{attribute 'linkalways'} 
{attribute 'no_explicit_call' := 'This FB is a CLASS and must be accessed using methods or properties'}
{attribute 'enable_dynamic_creation'}
FUNCTION_BLOCK NodeAddedEvent EXTENDS Disposable IMPLEMENTS I_NodeAddedEvent
VAR
	_target : I_Node;
END_VAR

METHOD FB_init : BOOL
VAR_INPUT
	bInitRetains : BOOL; // if TRUE, the retain variables are initialized (warm start / cold start)
	bInCopyCode : BOOL;  // if TRUE, the instance afterwards gets moved into the copy code (online change)
	Target : I_Node;
END_VAR
This^._target := Target;
END_METHOD

PROPERTY PUBLIC Target : I_Node
GET
Target := _target;
END_GET
END_PROPERTY

END_FUNCTION_BLOCK

(* stored: Version 1.1.0.1, ProductVersion 3.1.4024.12
   POU NodeAddedEvent: Id {675de5f9-7ea0-47ea-9f02-f8d732921215}, SpecialFunc None
   Folder Constructor: Id {3f775415-77de-4978-87d9-9c8a995c1d0f}
   Method FB_init: Id {79ddcdd9-31d4-44ed-94b0-7a9f63d0fbef}
   Property Target: Id {4a2bcc78-f497-4e83-a8f4-9474f407e865}
   Get Get: Id {d31b74b6-af7f-4406-80fa-20b002fddf8b} *)
